{attribute 'qualified_only'}
VAR_GLOBAL
	i_UltrasonicSensor AT %I* : INT;
	i_voltageUltrasonicSensor AT %Q* : INT;
	r_bufferUltraschall : ARRAY [1..100] OF REAL;
END_VAR

(* stored: Version 1.1.0.1, ProductVersion 3.1.4022.12
   GVL GVL: Id {abac1db7-5ebb-4cb1-bcc2-f9bea12053ed} *)
